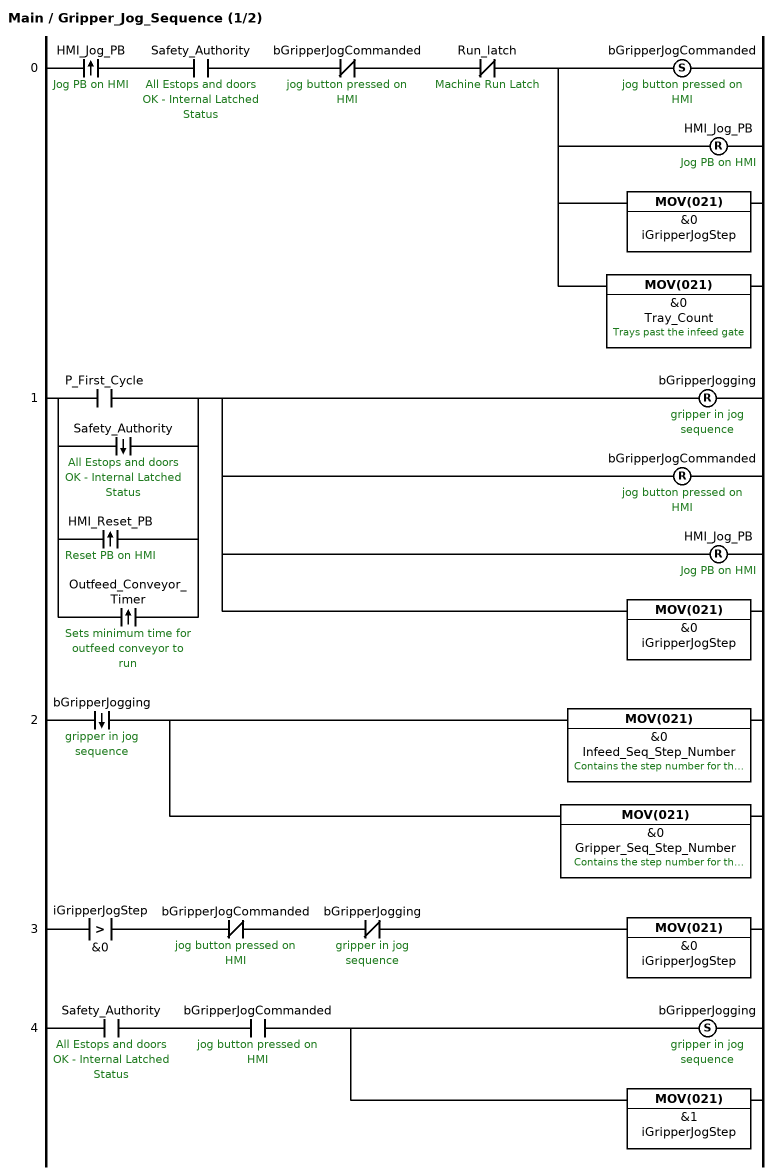
; [picture p144: Main / Gripper_Jog_Sequence, rungs 0-4]
; rung 0
@LD HMI_Jog_PB  ; Jog PB on HMI
AND Safety_Authority  ; All Estops and doors OK - Internal Latched Status
ANDNOT bGripperJogCommanded  ; jog button pressed on HMI
ANDNOT Run_latch  ; Machine Run Latch
SET bGripperJogCommanded  ; jog button pressed on HMI
RSET HMI_Jog_PB  ; Jog PB on HMI
MOV(021) &0 iGripperJogStep
MOV(021) &0 Tray_Count  ; Trays past the infeed gate
; rung 1
LD P_First_Cycle
%OR Safety_Authority  ; All Estops and doors OK - Internal Latched Status
@OR HMI_Reset_PB  ; Reset PB on HMI
@OR Outfeed_Conveyor_Timer  ; Sets minimum time for outfeed conveyor to run
RSET bGripperJogging  ; gripper in jog sequence
RSET bGripperJogCommanded  ; jog button pressed on HMI
RSET HMI_Jog_PB  ; Jog PB on HMI
MOV(021) &0 iGripperJogStep
; rung 2
%LD bGripperJogging  ; gripper in jog sequence
MOV(021) &0 Infeed_Seq_Step_Number  ; Contains the step number for the Infeed sequence
MOV(021) &0 Gripper_Seq_Step_Number  ; Contains the step number for the gripper sequence
; rung 3
LD>(320) iGripperJogStep &0
ANDNOT bGripperJogCommanded  ; jog button pressed on HMI
ANDNOT bGripperJogging  ; gripper in jog sequence
MOV(021) &0 iGripperJogStep
; rung 4
LD Safety_Authority  ; All Estops and doors OK - Internal Latched Status
AND bGripperJogCommanded  ; jog button pressed on HMI
SET bGripperJogging  ; gripper in jog sequence
MOV(021) &1 iGripperJogStep

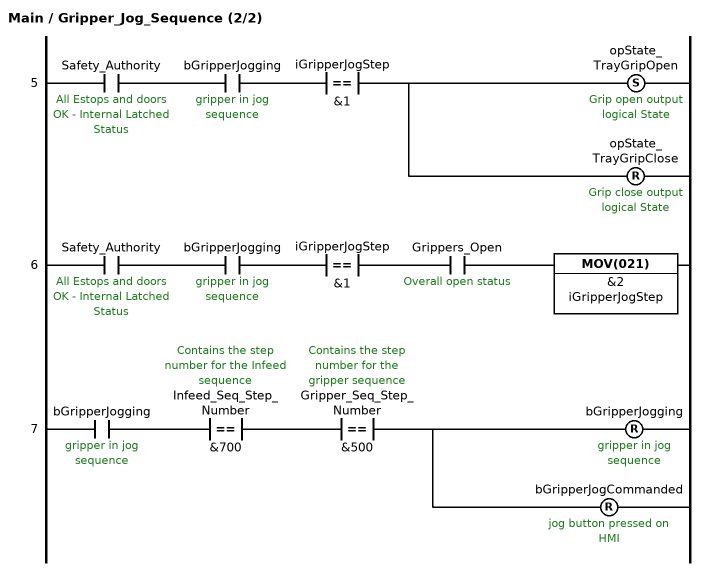
; rung 5
LD Safety_Authority  ; All Estops and doors OK - Internal Latched Status
AND bGripperJogging  ; gripper in jog sequence
AND=(300) iGripperJogStep &1
SET opState_TrayGripOpen  ; Grip open output logical State
RSET opState_TrayGripClose  ; Grip close output logical State
; rung 6
LD Safety_Authority  ; All Estops and doors OK - Internal Latched Status
AND bGripperJogging  ; gripper in jog sequence
AND=(300) iGripperJogStep &1
AND Grippers_Open  ; Overall open status
MOV(021) &2 iGripperJogStep
; rung 7
LD bGripperJogging  ; gripper in jog sequence
AND=(300) Infeed_Seq_Step_Number &700  ; Contains the step number for the Infeed sequence
AND=(300) Gripper_Seq_Step_Number &500  ; Contains the step number for the gripper sequence
RSET bGripperJogging  ; gripper in jog sequence
RSET bGripperJogCommanded  ; jog button pressed on HMI

### Section Machine_Timing

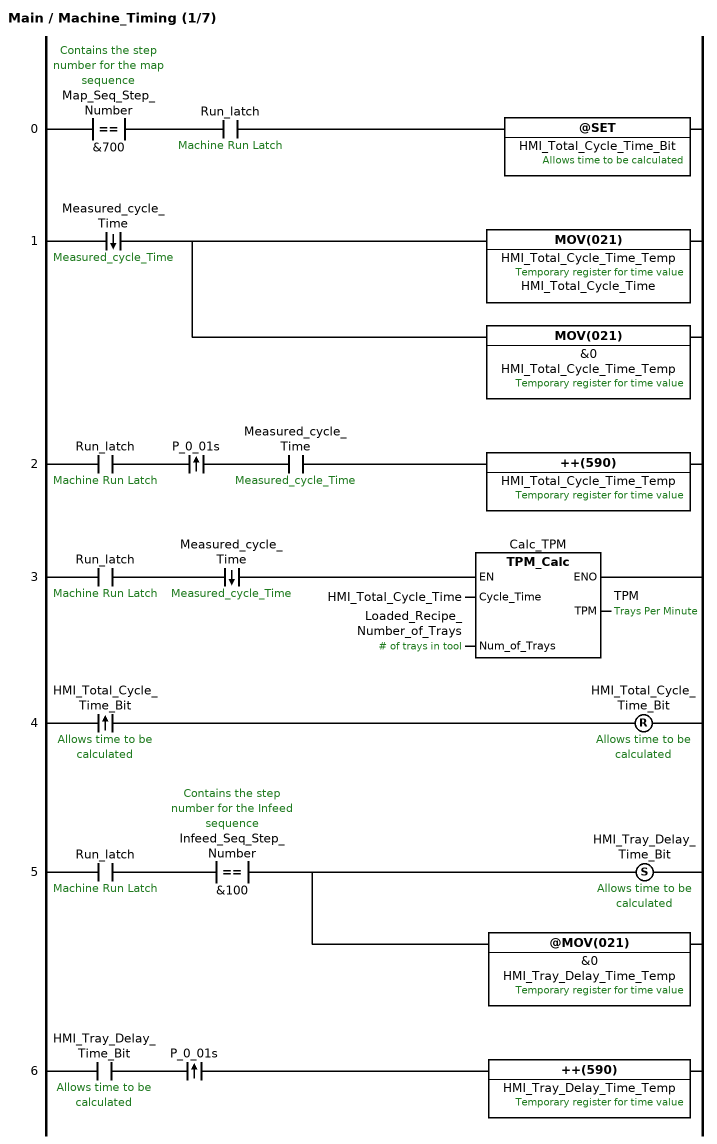
; rung 0
LD=(300) Map_Seq_Step_Number &700  ; Contains the step number for the map sequence
AND Run_latch  ; Machine Run Latch
@SET HMI_Total_Cycle_Time_Bit  ; Allows time to be calculated
; rung 1
%LD Measured_cycle_Time  ; Measured_cycle_Time
MOV(021) HMI_Total_Cycle_Time_Temp HMI_Total_Cycle_Time  ; Temporary register for time value
MOV(021) &0 HMI_Total_Cycle_Time_Temp  ; Temporary register for time value
; rung 2
LD Run_latch  ; Machine Run Latch
@AND P_0_01s
AND Measured_cycle_Time  ; Measured_cycle_Time
++(590) HMI_Total_Cycle_Time_Temp  ; Temporary register for time value
; rung 3
LD Run_latch  ; Machine Run Latch
%AND Measured_cycle_Time  ; Measured_cycle_Time
CALL Calc_TPM : TPM_Calc (Cycle_Time := HMI_Total_Cycle_Time, Num_of_Trays := Loaded_Recipe_Number_of_Trays, TPM => TPM)  ; # of trays in tool, Trays Per Minute
; rung 4
@LD HMI_Total_Cycle_Time_Bit  ; Allows time to be calculated
RSET HMI_Total_Cycle_Time_Bit  ; Allows time to be calculated
; rung 5
LD Run_latch  ; Machine Run Latch
AND=(300) Infeed_Seq_Step_Number &100  ; Contains the step number for the Infeed sequence
SET HMI_Tray_Delay_Time_Bit  ; Allows time to be calculated
@MOV(021) &0 HMI_Tray_Delay_Time_Temp  ; Temporary register for time value
; rung 6
LD HMI_Tray_Delay_Time_Bit  ; Allows time to be calculated
@AND P_0_01s
++(590) HMI_Tray_Delay_Time_Temp  ; Temporary register for time value

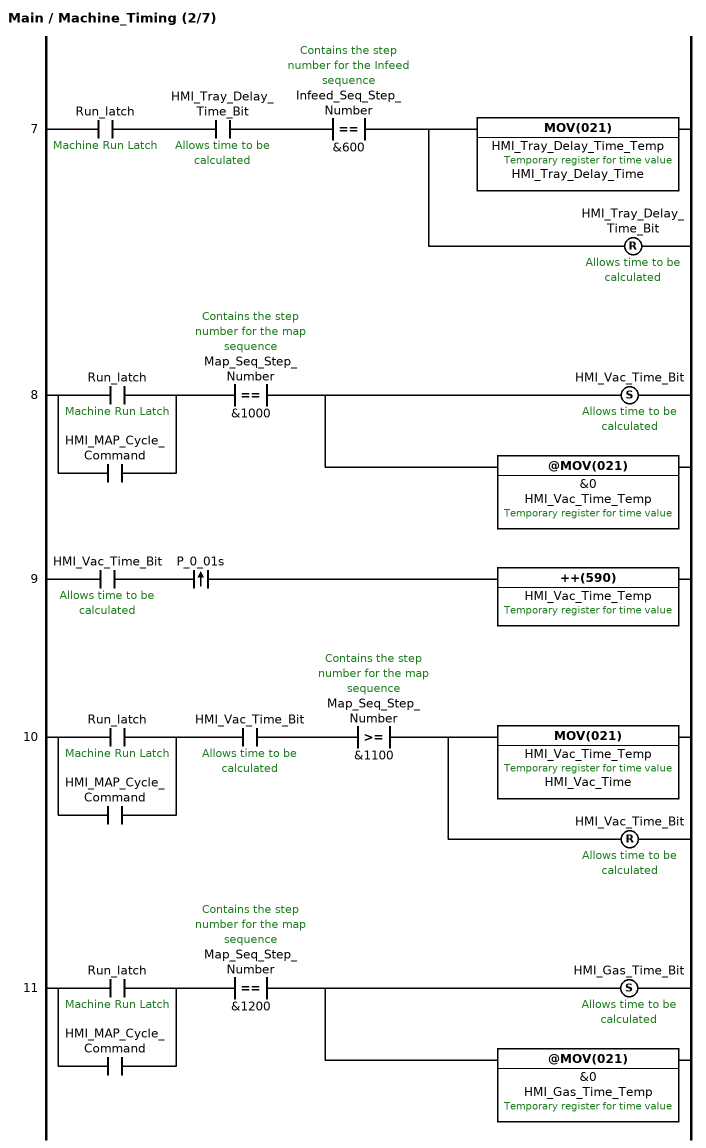
; rung 7
LD Run_latch  ; Machine Run Latch
AND HMI_Tray_Delay_Time_Bit  ; Allows time to be calculated
AND=(300) Infeed_Seq_Step_Number &600  ; Contains the step number for the Infeed sequence
MOV(021) HMI_Tray_Delay_Time_Temp HMI_Tray_Delay_Time  ; Temporary register for time value
RSET HMI_Tray_Delay_Time_Bit  ; Allows time to be calculated
; rung 8
LD Run_latch  ; Machine Run Latch
OR HMI_MAP_Cycle_Command
AND=(300) Map_Seq_Step_Number &1000  ; Contains the step number for the map sequence
SET HMI_Vac_Time_Bit  ; Allows time to be calculated
@MOV(021) &0 HMI_Vac_Time_Temp  ; Temporary register for time value
; rung 9
LD HMI_Vac_Time_Bit  ; Allows time to be calculated
@AND P_0_01s
++(590) HMI_Vac_Time_Temp  ; Temporary register for time value
; rung 10
LD Run_latch  ; Machine Run Latch
OR HMI_MAP_Cycle_Command
AND HMI_Vac_Time_Bit  ; Allows time to be calculated
AND>=(325) Map_Seq_Step_Number &1100  ; Contains the step number for the map sequence
MOV(021) HMI_Vac_Time_Temp HMI_Vac_Time  ; Temporary register for time value
RSET HMI_Vac_Time_Bit  ; Allows time to be calculated
; rung 11
LD Run_latch  ; Machine Run Latch
OR HMI_MAP_Cycle_Command
AND=(300) Map_Seq_Step_Number &1200  ; Contains the step number for the map sequence
SET HMI_Gas_Time_Bit  ; Allows time to be calculated
@MOV(021) &0 HMI_Gas_Time_Temp  ; Temporary register for time value

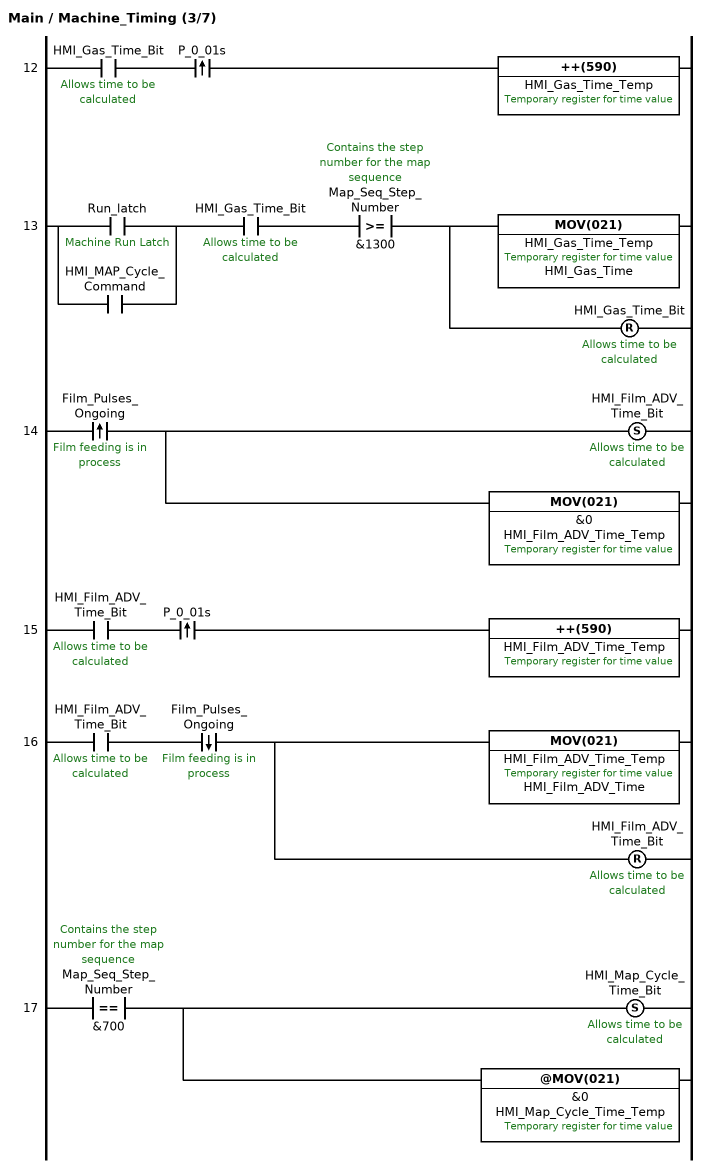
; rung 12
LD HMI_Gas_Time_Bit  ; Allows time to be calculated
@AND P_0_01s
++(590) HMI_Gas_Time_Temp  ; Temporary register for time value
; rung 13
LD Run_latch  ; Machine Run Latch
OR HMI_MAP_Cycle_Command
AND HMI_Gas_Time_Bit  ; Allows time to be calculated
AND>=(325) Map_Seq_Step_Number &1300  ; Contains the step number for the map sequence
MOV(021) HMI_Gas_Time_Temp HMI_Gas_Time  ; Temporary register for time value
RSET HMI_Gas_Time_Bit  ; Allows time to be calculated
; rung 14
@LD Film_Pulses_Ongoing  ; Film feeding is in process
SET HMI_Film_ADV_Time_Bit  ; Allows time to be calculated
MOV(021) &0 HMI_Film_ADV_Time_Temp  ; Temporary register for time value
; rung 15
LD HMI_Film_ADV_Time_Bit  ; Allows time to be calculated
@AND P_0_01s
++(590) HMI_Film_ADV_Time_Temp  ; Temporary register for time value
; rung 16
LD HMI_Film_ADV_Time_Bit  ; Allows time to be calculated
%AND Film_Pulses_Ongoing  ; Film feeding is in process
MOV(021) HMI_Film_ADV_Time_Temp HMI_Film_ADV_Time  ; Temporary register for time value
RSET HMI_Film_ADV_Time_Bit  ; Allows time to be calculated
; rung 17
LD=(300) Map_Seq_Step_Number &700  ; Contains the step number for the map sequence
SET HMI_Map_Cycle_Time_Bit  ; Allows time to be calculated
@MOV(021) &0 HMI_Map_Cycle_Time_Temp  ; Temporary register for time value

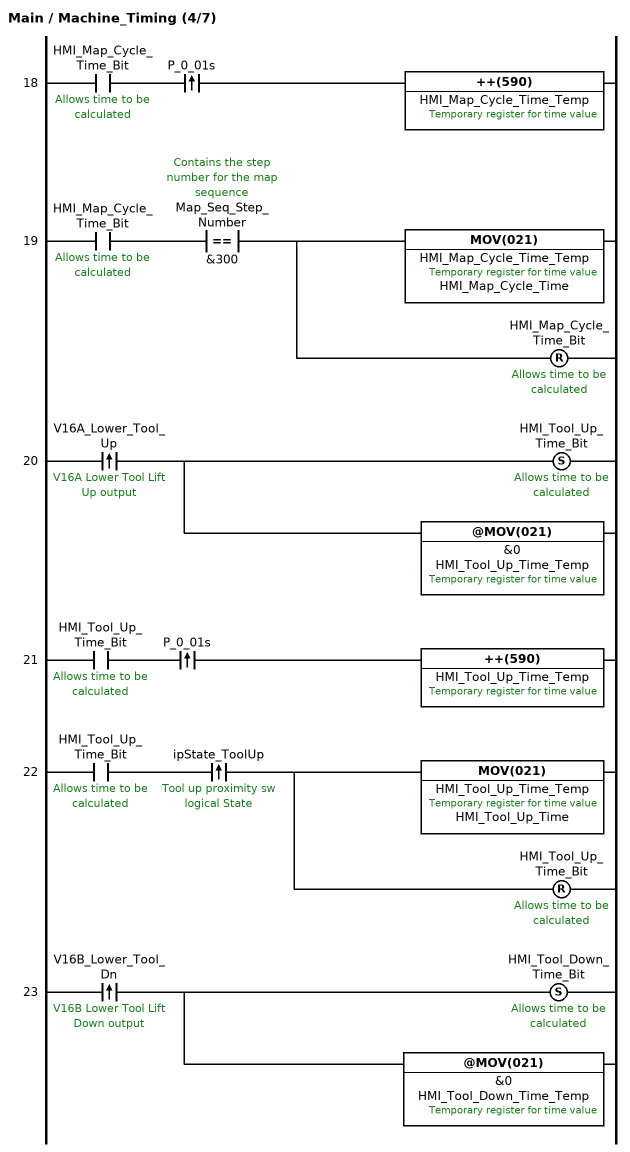
; rung 18
LD HMI_Map_Cycle_Time_Bit  ; Allows time to be calculated
@AND P_0_01s
++(590) HMI_Map_Cycle_Time_Temp  ; Temporary register for time value
; rung 19
LD HMI_Map_Cycle_Time_Bit  ; Allows time to be calculated
AND=(300) Map_Seq_Step_Number &300  ; Contains the step number for the map sequence
MOV(021) HMI_Map_Cycle_Time_Temp HMI_Map_Cycle_Time  ; Temporary register for time value
RSET HMI_Map_Cycle_Time_Bit  ; Allows time to be calculated
; rung 20
@LD V16A_Lower_Tool_Up  ; V16A Lower Tool Lift Up output
SET HMI_Tool_Up_Time_Bit  ; Allows time to be calculated
@MOV(021) &0 HMI_Tool_Up_Time_Temp  ; Temporary register for time value
; rung 21
LD HMI_Tool_Up_Time_Bit  ; Allows time to be calculated
@AND P_0_01s
++(590) HMI_Tool_Up_Time_Temp  ; Temporary register for time value
; rung 22
LD HMI_Tool_Up_Time_Bit  ; Allows time to be calculated
@AND ipState_ToolUp  ; Tool up proximity sw logical State
MOV(021) HMI_Tool_Up_Time_Temp HMI_Tool_Up_Time  ; Temporary register for time value
RSET HMI_Tool_Up_Time_Bit  ; Allows time to be calculated
; rung 23
@LD V16B_Lower_Tool_Dn  ; V16B Lower Tool Lift Down output
SET HMI_Tool_Down_Time_Bit  ; Allows time to be calculated
@MOV(021) &0 HMI_Tool_Down_Time_Temp  ; Temporary register for time value

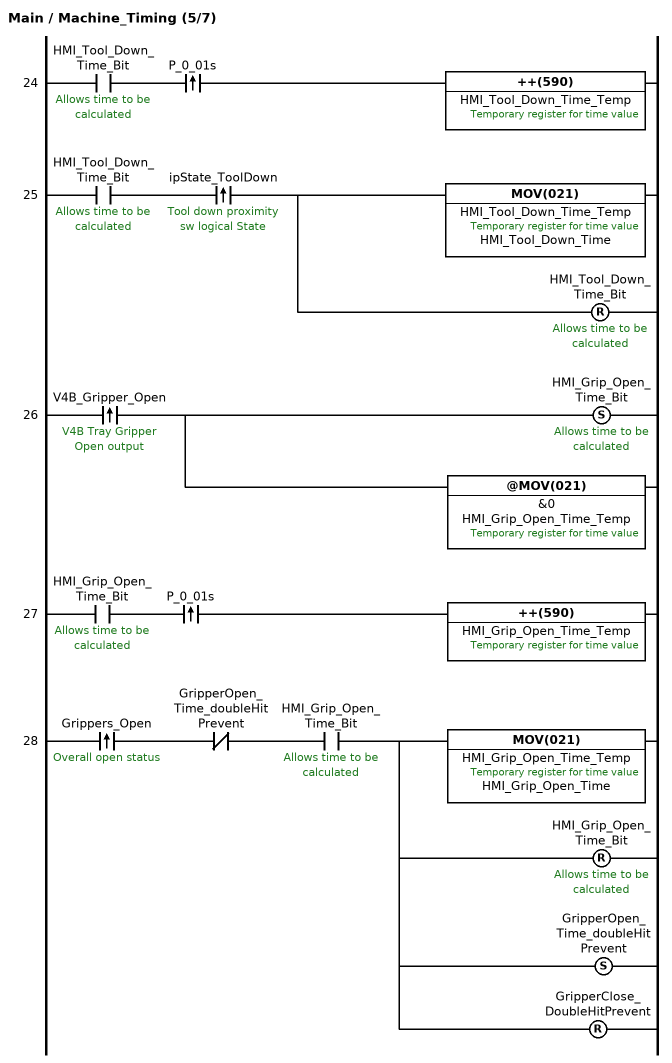
; rung 24
LD HMI_Tool_Down_Time_Bit  ; Allows time to be calculated
@AND P_0_01s
++(590) HMI_Tool_Down_Time_Temp  ; Temporary register for time value
; rung 25
LD HMI_Tool_Down_Time_Bit  ; Allows time to be calculated
@AND ipState_ToolDown  ; Tool down proximity sw logical State
MOV(021) HMI_Tool_Down_Time_Temp HMI_Tool_Down_Time  ; Temporary register for time value
RSET HMI_Tool_Down_Time_Bit  ; Allows time to be calculated
; rung 26
@LD V4B_Gripper_Open  ; V4B Tray Gripper Open output
SET HMI_Grip_Open_Time_Bit  ; Allows time to be calculated
@MOV(021) &0 HMI_Grip_Open_Time_Temp  ; Temporary register for time value
; rung 27
LD HMI_Grip_Open_Time_Bit  ; Allows time to be calculated
@AND P_0_01s
++(590) HMI_Grip_Open_Time_Temp  ; Temporary register for time value
; rung 28
@LD Grippers_Open  ; Overall open status
ANDNOT GripperOpen_Time_doubleHitPrevent
AND HMI_Grip_Open_Time_Bit  ; Allows time to be calculated
MOV(021) HMI_Grip_Open_Time_Temp HMI_Grip_Open_Time  ; Temporary register for time value
RSET HMI_Grip_Open_Time_Bit  ; Allows time to be calculated
SET GripperOpen_Time_doubleHitPrevent
RSET GripperClose_DoubleHitPrevent

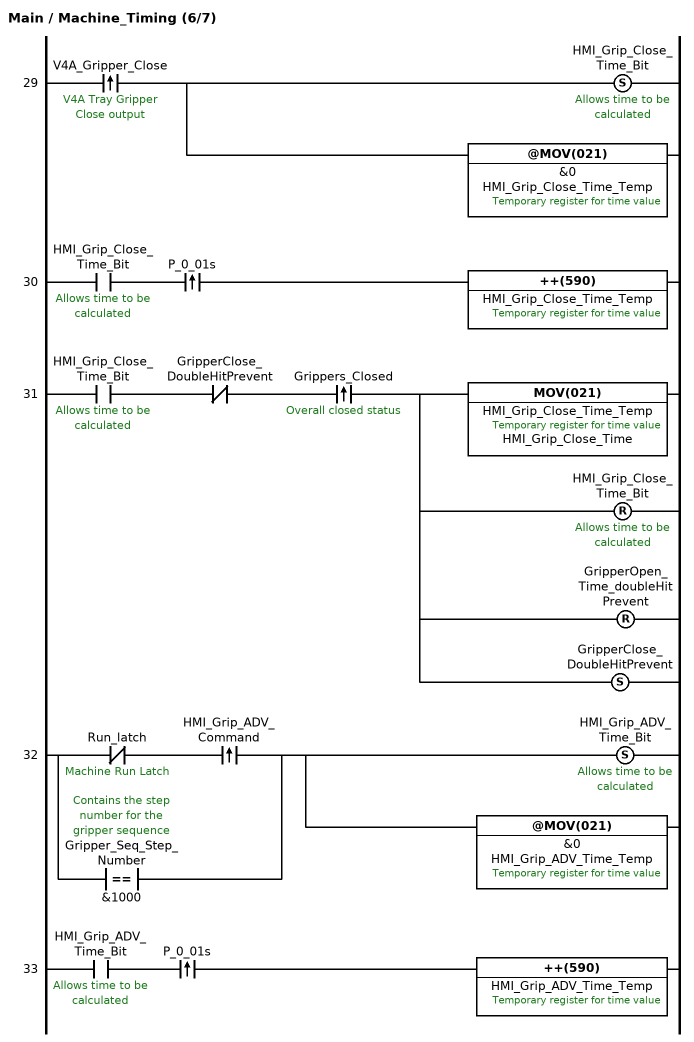
; rung 29
@LD V4A_Gripper_Close  ; V4A Tray Gripper Close output
SET HMI_Grip_Close_Time_Bit  ; Allows time to be calculated
@MOV(021) &0 HMI_Grip_Close_Time_Temp  ; Temporary register for time value
; rung 30
LD HMI_Grip_Close_Time_Bit  ; Allows time to be calculated
@AND P_0_01s
++(590) HMI_Grip_Close_Time_Temp  ; Temporary register for time value
; rung 31
LD HMI_Grip_Close_Time_Bit  ; Allows time to be calculated
ANDNOT GripperClose_DoubleHitPrevent
@AND Grippers_Closed  ; Overall closed status
MOV(021) HMI_Grip_Close_Time_Temp HMI_Grip_Close_Time  ; Temporary register for time value
RSET HMI_Grip_Close_Time_Bit  ; Allows time to be calculated
RSET GripperOpen_Time_doubleHitPrevent
SET GripperClose_DoubleHitPrevent
; rung 32
LDNOT Run_latch  ; Machine Run Latch
@AND HMI_Grip_ADV_Command
OR=(300) Gripper_Seq_Step_Number &1000  ; Contains the step number for the gripper sequence
SET HMI_Grip_ADV_Time_Bit  ; Allows time to be calculated
@MOV(021) &0 HMI_Grip_ADV_Time_Temp  ; Temporary register for time value
; rung 33
LD HMI_Grip_ADV_Time_Bit  ; Allows time to be calculated
@AND P_0_01s
++(590) HMI_Grip_ADV_Time_Temp  ; Temporary register for time value

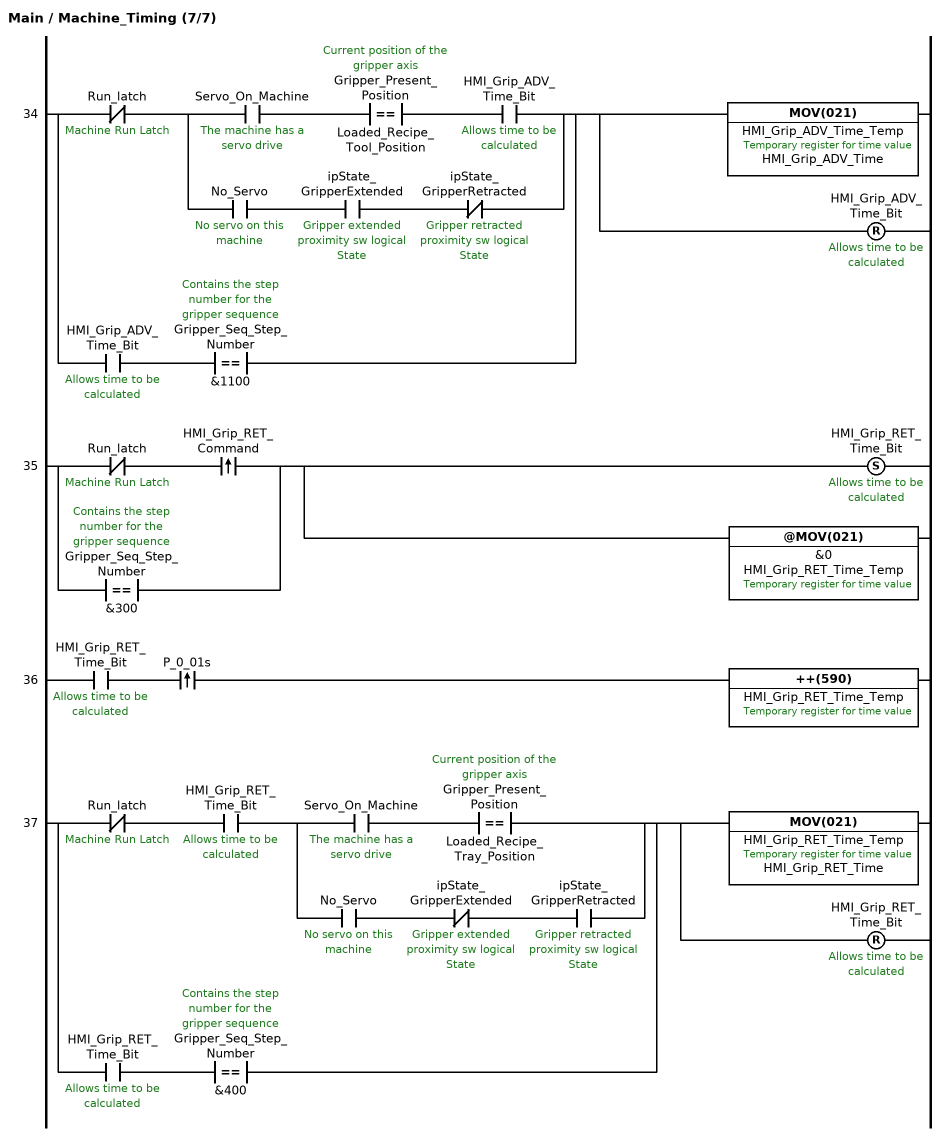
; rung 34
LDNOT Run_latch  ; Machine Run Latch
LD Servo_On_Machine  ; The machine has a servo drive
AND=(300) Gripper_Present_Position Loaded_Recipe_Tool_Position  ; Current position of the gripper axis
AND HMI_Grip_ADV_Time_Bit  ; Allows time to be calculated
LD No_Servo  ; No servo on this machine
AND ipState_GripperExtended  ; Gripper extended proximity sw logical State
ANDNOT ipState_GripperRetracted  ; Gripper retracted proximity sw logical State
ORLD
ANDLD
LD HMI_Grip_ADV_Time_Bit  ; Allows time to be calculated
AND=(300) Gripper_Seq_Step_Number &1100  ; Contains the step number for the gripper sequence
ORLD
MOV(021) HMI_Grip_ADV_Time_Temp HMI_Grip_ADV_Time  ; Temporary register for time value
RSET HMI_Grip_ADV_Time_Bit  ; Allows time to be calculated
; rung 35
LDNOT Run_latch  ; Machine Run Latch
@AND HMI_Grip_RET_Command
OR=(300) Gripper_Seq_Step_Number &300  ; Contains the step number for the gripper sequence
SET HMI_Grip_RET_Time_Bit  ; Allows time to be calculated
@MOV(021) &0 HMI_Grip_RET_Time_Temp  ; Temporary register for time value
; rung 36
LD HMI_Grip_RET_Time_Bit  ; Allows time to be calculated
@AND P_0_01s
++(590) HMI_Grip_RET_Time_Temp  ; Temporary register for time value
; rung 37
LDNOT Run_latch  ; Machine Run Latch
AND HMI_Grip_RET_Time_Bit  ; Allows time to be calculated
LD Servo_On_Machine  ; The machine has a servo drive
AND=(300) Gripper_Present_Position Loaded_Recipe_Tray_Position  ; Current position of the gripper axis
LD No_Servo  ; No servo on this machine
ANDNOT ipState_GripperExtended  ; Gripper extended proximity sw logical State
AND ipState_GripperRetracted  ; Gripper retracted proximity sw logical State
ORLD
ANDLD
LD HMI_Grip_RET_Time_Bit  ; Allows time to be calculated
AND=(300) Gripper_Seq_Step_Number &400  ; Contains the step number for the gripper sequence
ORLD
MOV(021) HMI_Grip_RET_Time_Temp HMI_Grip_RET_Time  ; Temporary register for time value
RSET HMI_Grip_RET_Time_Bit  ; Allows time to be calculated

### Section Vacuum_Test

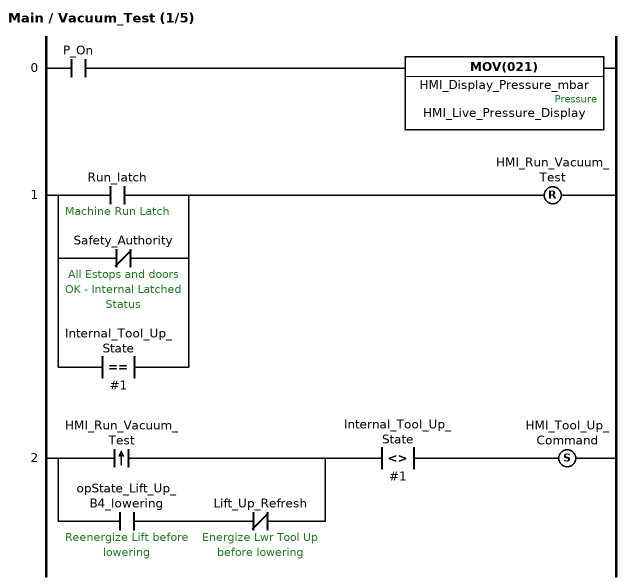
; rung 0
LD P_On
MOV(021) HMI_Display_Pressure_mbar HMI_Live_Pressure_Display  ; Pressure
; rung 1
LD Run_latch  ; Machine Run Latch
ORNOT Safety_Authority  ; All Estops and doors OK - Internal Latched Status
OR=(300) Internal_Tool_Up_State #1
RSET HMI_Run_Vacuum_Test
; rung 2
@LD HMI_Run_Vacuum_Test
LD opState_Lift_Up_B4_lowering  ; Reenergize Lift before lowering
ANDNOT Lift_Up_Refresh  ; Energize Lwr Tool Up before lowering
ORLD
AND<>(305) Internal_Tool_Up_State #1
SET HMI_Tool_Up_Command

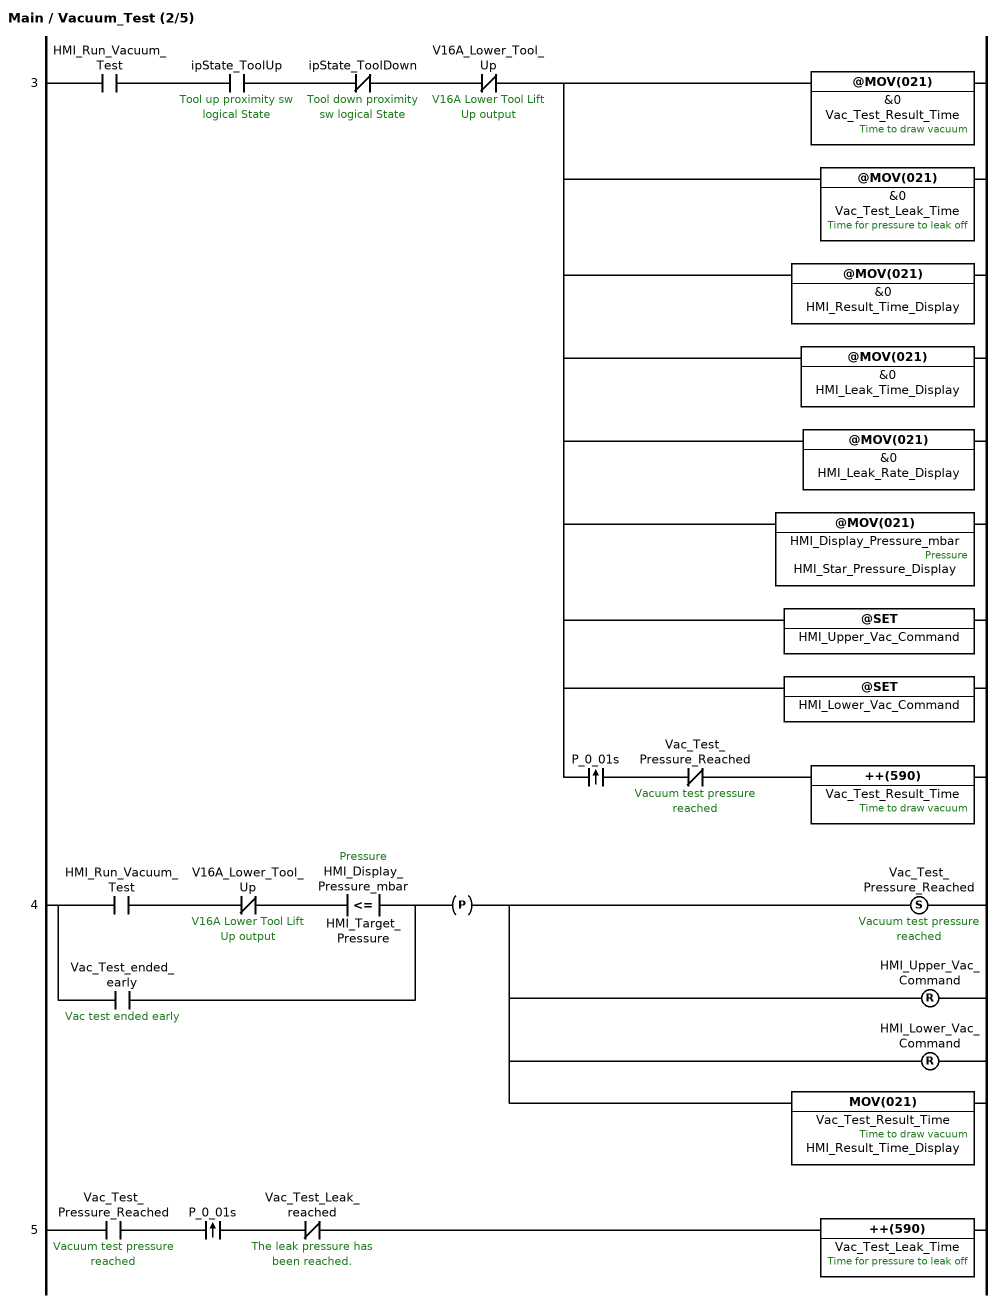
; rung 3
LD HMI_Run_Vacuum_Test
AND ipState_ToolUp  ; Tool up proximity sw logical State
ANDNOT ipState_ToolDown  ; Tool down proximity sw logical State
ANDNOT V16A_Lower_Tool_Up  ; V16A Lower Tool Lift Up output
@MOV(021) &0 Vac_Test_Result_Time  ; Time to draw vacuum
@MOV(021) &0 Vac_Test_Leak_Time  ; Time for pressure to leak off
@MOV(021) &0 HMI_Result_Time_Display
@MOV(021) &0 HMI_Leak_Time_Display
@MOV(021) &0 HMI_Leak_Rate_Display
@MOV(021) HMI_Display_Pressure_mbar HMI_Star_Pressure_Display  ; Pressure
@SET HMI_Upper_Vac_Command
@SET HMI_Lower_Vac_Command
@AND P_0_01s
ANDNOT Vac_Test_Pressure_Reached  ; Vacuum test pressure reached
++(590) Vac_Test_Result_Time  ; Time to draw vacuum
; rung 4
LD HMI_Run_Vacuum_Test
ANDNOT V16A_Lower_Tool_Up  ; V16A Lower Tool Lift Up output
AND<=(315) HMI_Display_Pressure_mbar HMI_Target_Pressure  ; Pressure
OR Vac_Test_ended_early  ; Vac test ended early
UP(521)
SET Vac_Test_Pressure_Reached  ; Vacuum test pressure reached
RSET HMI_Upper_Vac_Command
RSET HMI_Lower_Vac_Command
MOV(021) Vac_Test_Result_Time HMI_Result_Time_Display  ; Time to draw vacuum
; rung 5
LD Vac_Test_Pressure_Reached  ; Vacuum test pressure reached
@AND P_0_01s
ANDNOT Vac_Test_Leak_reached  ; The leak pressure has been reached.
++(590) Vac_Test_Leak_Time  ; Time for pressure to leak off

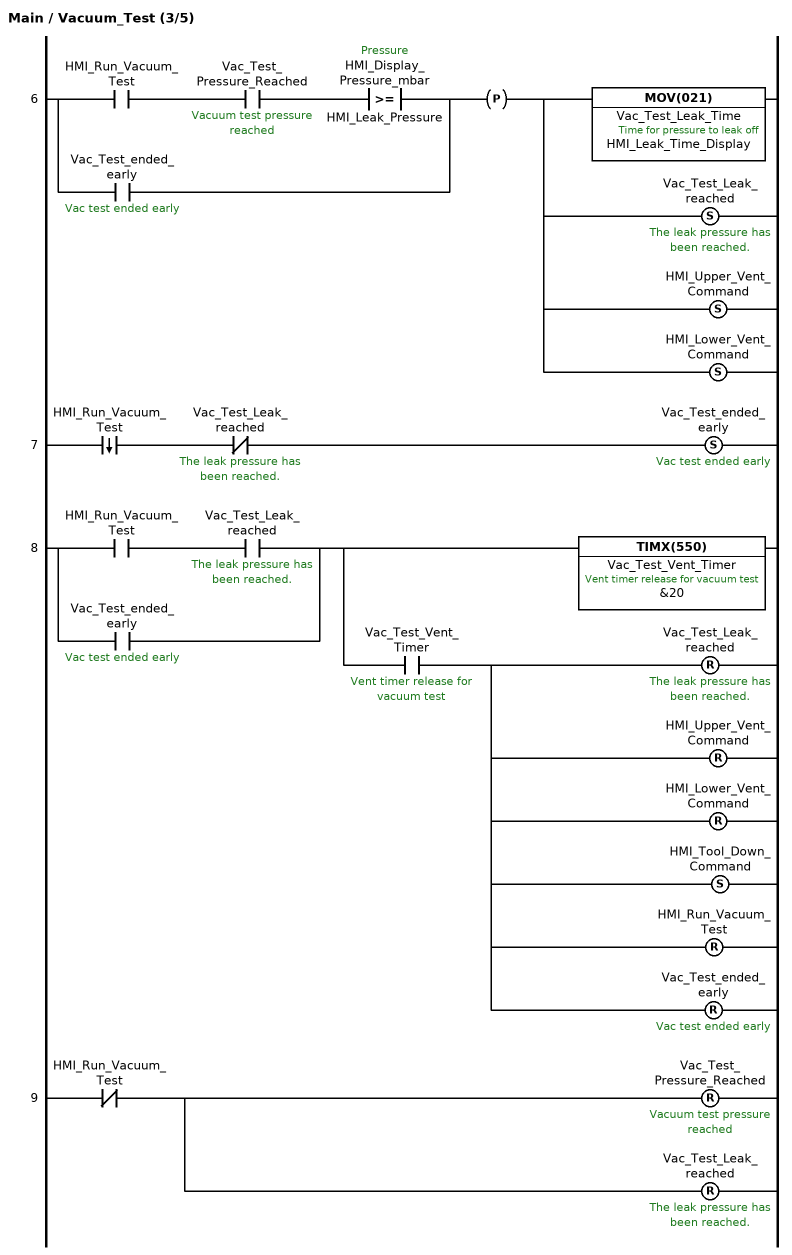
; rung 6
LD HMI_Run_Vacuum_Test
AND Vac_Test_Pressure_Reached  ; Vacuum test pressure reached
AND>=(325) HMI_Display_Pressure_mbar HMI_Leak_Pressure  ; Pressure
OR Vac_Test_ended_early  ; Vac test ended early
UP(521)
MOV(021) Vac_Test_Leak_Time HMI_Leak_Time_Display  ; Time for pressure to leak off
SET Vac_Test_Leak_reached  ; The leak pressure has been reached.
SET HMI_Upper_Vent_Command
SET HMI_Lower_Vent_Command
; rung 7
%LD HMI_Run_Vacuum_Test
ANDNOT Vac_Test_Leak_reached  ; The leak pressure has been reached.
SET Vac_Test_ended_early  ; Vac test ended early
; rung 8
LD HMI_Run_Vacuum_Test
AND Vac_Test_Leak_reached  ; The leak pressure has been reached.
OR Vac_Test_ended_early  ; Vac test ended early
TIMX(550) Vac_Test_Vent_Timer &20  ; Vent timer release for vacuum test
AND Vac_Test_Vent_Timer  ; Vent timer release for vacuum test
RSET Vac_Test_Leak_reached  ; The leak pressure has been reached.
RSET HMI_Upper_Vent_Command
RSET HMI_Lower_Vent_Command
SET HMI_Tool_Down_Command
RSET HMI_Run_Vacuum_Test
RSET Vac_Test_ended_early  ; Vac test ended early
; rung 9
LDNOT HMI_Run_Vacuum_Test
RSET Vac_Test_Pressure_Reached  ; Vacuum test pressure reached
RSET Vac_Test_Leak_reached  ; The leak pressure has been reached.

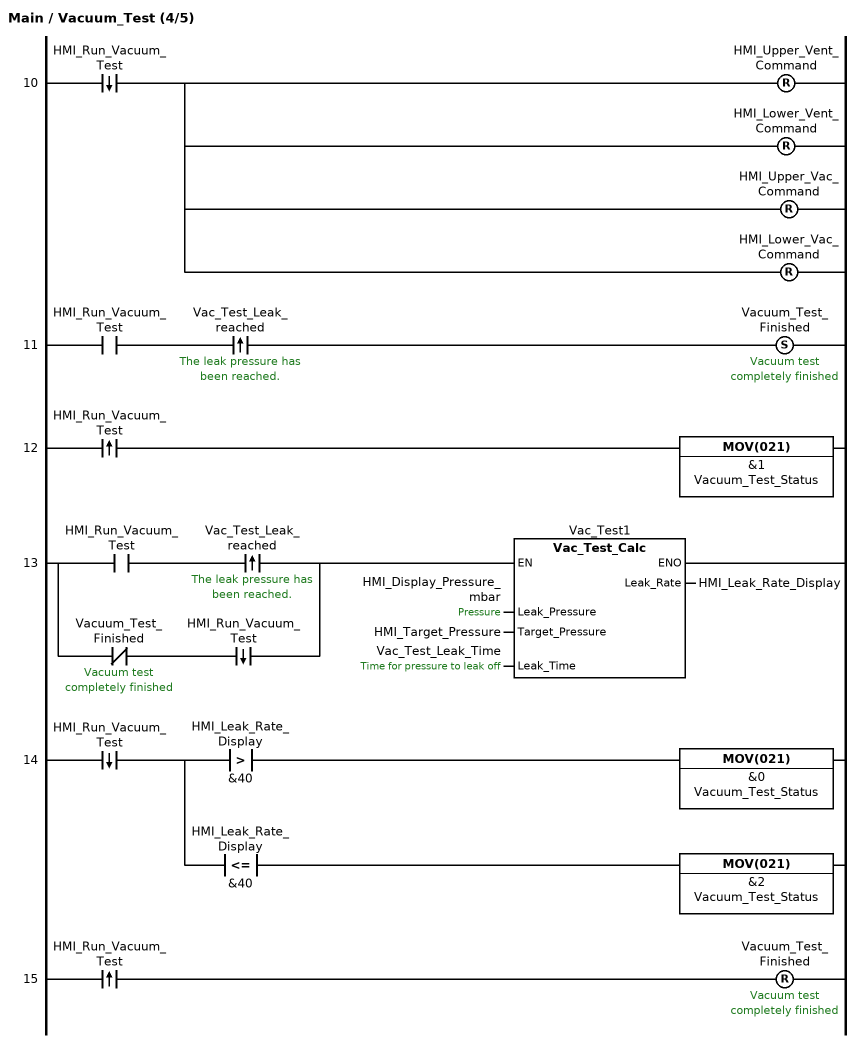
; rung 10
%LD HMI_Run_Vacuum_Test
RSET HMI_Upper_Vent_Command
RSET HMI_Lower_Vent_Command
RSET HMI_Upper_Vac_Command
RSET HMI_Lower_Vac_Command
; rung 11
LD HMI_Run_Vacuum_Test
@AND Vac_Test_Leak_reached  ; The leak pressure has been reached.
SET Vacuum_Test_Finished  ; Vacuum test completely finished
; rung 12
@LD HMI_Run_Vacuum_Test
MOV(021) &1 Vacuum_Test_Status
; rung 13
LD HMI_Run_Vacuum_Test
@AND Vac_Test_Leak_reached  ; The leak pressure has been reached.
LDNOT Vacuum_Test_Finished  ; Vacuum test completely finished
%AND HMI_Run_Vacuum_Test
ORLD
CALL Vac_Test1 : Vac_Test_Calc (Leak_Pressure := HMI_Display_Pressure_mbar, Target_Pressure := HMI_Target_Pressure, Leak_Time := Vac_Test_Leak_Time, Leak_Rate => HMI_Leak_Rate_Display)  ; Pressure, Time for pressure to leak off
; rung 14
%LD HMI_Run_Vacuum_Test
OUT TR0
AND>(320) HMI_Leak_Rate_Display &40
MOV(021) &0 Vacuum_Test_Status
LD TR0
AND<=(315) HMI_Leak_Rate_Display &40
MOV(021) &2 Vacuum_Test_Status
; rung 15
@LD HMI_Run_Vacuum_Test
RSET Vacuum_Test_Finished  ; Vacuum test completely finished

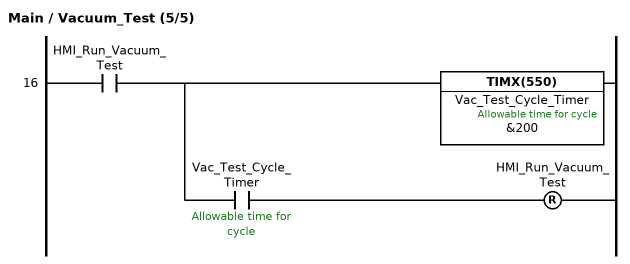
; rung 16
LD HMI_Run_Vacuum_Test
TIMX(550) Vac_Test_Cycle_Timer &200  ; Allowable time for cycle
AND Vac_Test_Cycle_Timer  ; Allowable time for cycle
RSET HMI_Run_Vacuum_Test

### Section HMI

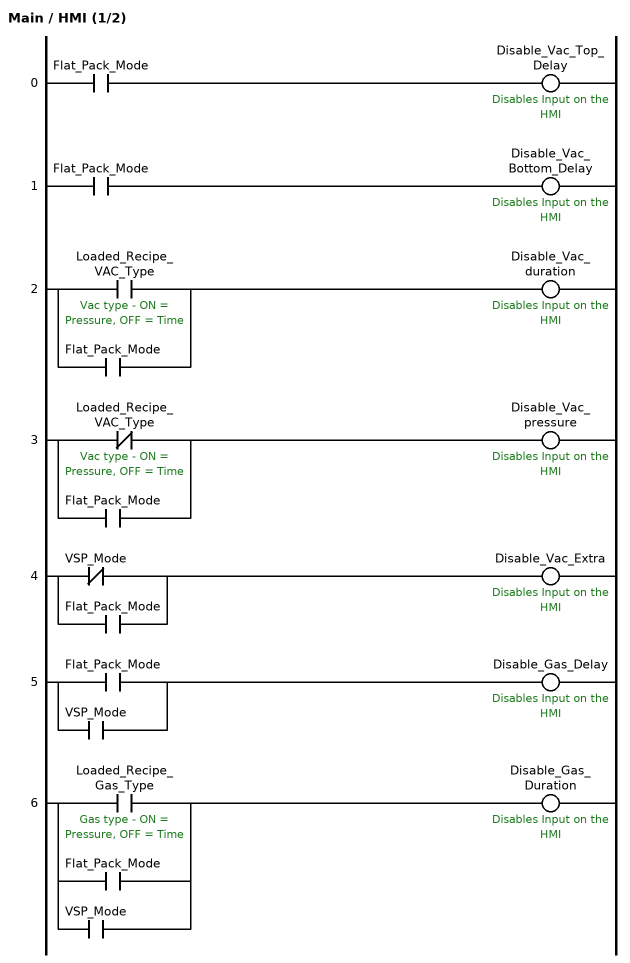
; rung 0
LD Flat_Pack_Mode
OUT Disable_Vac_Top_Delay  ; Disables Input on the HMI
; rung 1
LD Flat_Pack_Mode
OUT Disable_Vac_Bottom_Delay  ; Disables Input on the HMI
; rung 2
LD Loaded_Recipe_VAC_Type  ; Vac type - ON = Pressure, OFF = Time
OR Flat_Pack_Mode
OUT Disable_Vac_duration  ; Disables Input on the HMI
; rung 3
LDNOT Loaded_Recipe_VAC_Type  ; Vac type - ON = Pressure, OFF = Time
OR Flat_Pack_Mode
OUT Disable_Vac_pressure  ; Disables Input on the HMI
; rung 4
LDNOT VSP_Mode
OR Flat_Pack_Mode
OUT Disable_Vac_Extra  ; Disables Input on the HMI
; rung 5
LD Flat_Pack_Mode
OR VSP_Mode
OUT Disable_Gas_Delay  ; Disables Input on the HMI
; rung 6
LD Loaded_Recipe_Gas_Type  ; Gas type - ON = Pressure, OFF = Time
OR Flat_Pack_Mode
OR VSP_Mode
OUT Disable_Gas_Duration  ; Disables Input on the HMI

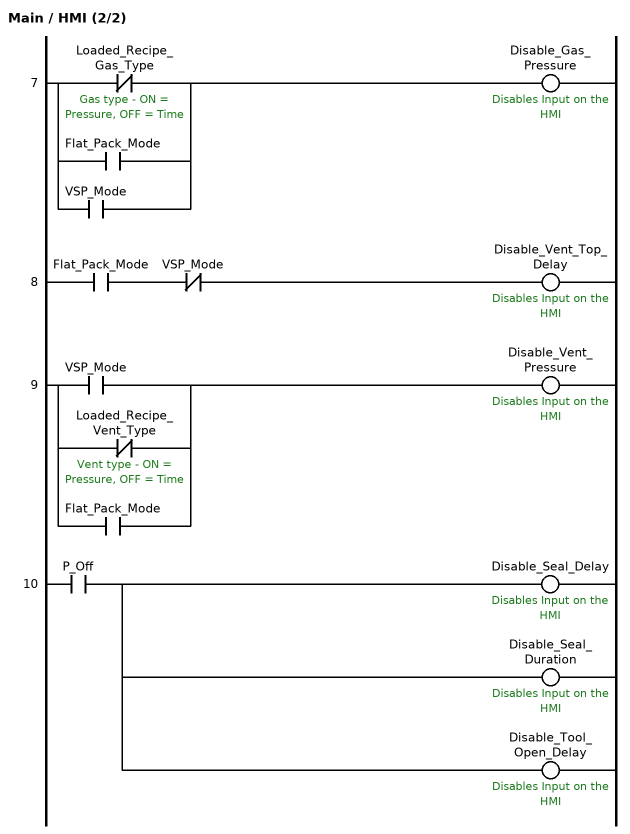
; rung 7
LDNOT Loaded_Recipe_Gas_Type  ; Gas type - ON = Pressure, OFF = Time
OR Flat_Pack_Mode
OR VSP_Mode
OUT Disable_Gas_Pressure  ; Disables Input on the HMI
; rung 8
LD Flat_Pack_Mode
ANDNOT VSP_Mode
OUT Disable_Vent_Top_Delay  ; Disables Input on the HMI
; rung 9
LD VSP_Mode
ORNOT Loaded_Recipe_Vent_Type  ; Vent type - ON = Pressure, OFF = Time
OR Flat_Pack_Mode
OUT Disable_Vent_Pressure  ; Disables Input on the HMI
; rung 10
LD P_Off
OUT Disable_Seal_Delay  ; Disables Input on the HMI
OUT Disable_Seal_Duration  ; Disables Input on the HMI
OUT Disable_Tool_Open_Delay  ; Disables Input on the HMI

### Section Vacuum_Graph

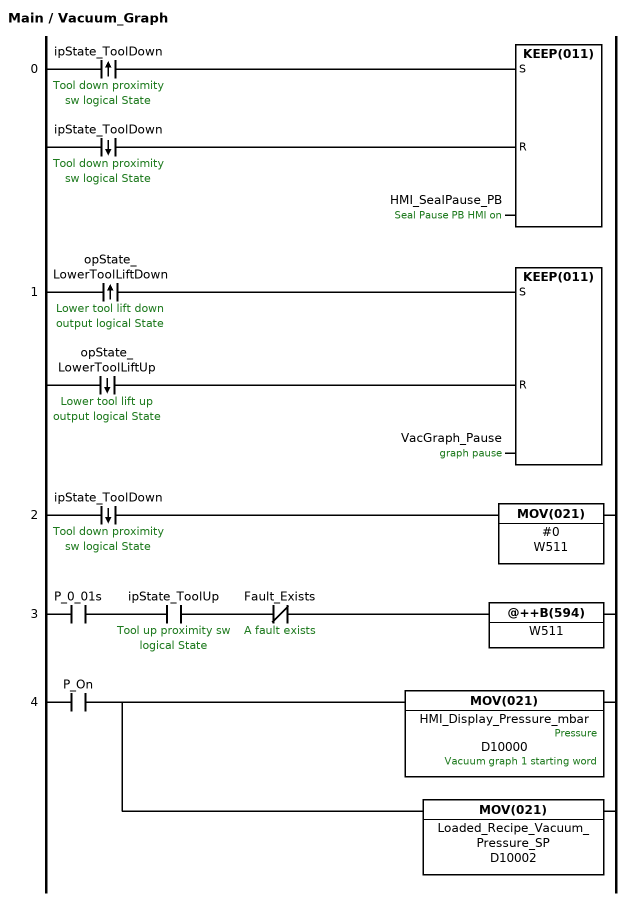
; rung 0
@LD ipState_ToolDown  ; Tool down proximity sw logical State
%LD ipState_ToolDown  ; Tool down proximity sw logical State
KEEP(011) HMI_SealPause_PB  ; Seal Pause PB HMI on
; rung 1
@LD opState_LowerToolLiftDown  ; Lower tool lift down output logical State
%LD opState_LowerToolLiftUp  ; Lower tool lift up output logical State
KEEP(011) VacGraph_Pause  ; graph pause
; rung 2
%LD ipState_ToolDown  ; Tool down proximity sw logical State
MOV(021) #0 W511
; rung 3
LD P_0_01s
AND ipState_ToolUp  ; Tool up proximity sw logical State
ANDNOT Fault_Exists  ; A fault exists
@++B(594) W511
; rung 4
LD P_On
MOV(021) HMI_Display_Pressure_mbar D10000  ; Pressure, Vacuum graph 1 starting word
MOV(021) Loaded_Recipe_Vacuum_Pressure_SP D10002

### Section PopUp

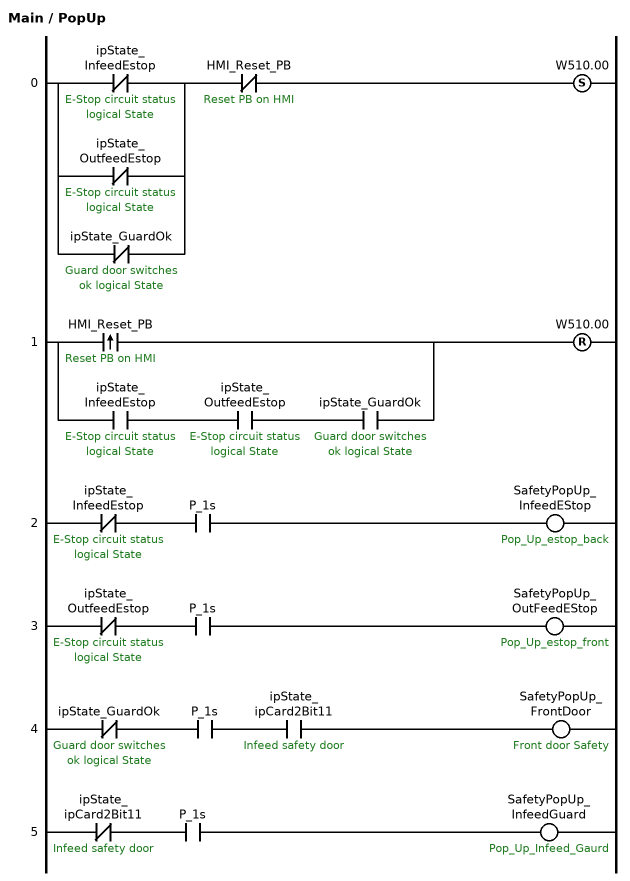
; rung 0
LDNOT ipState_InfeedEstop  ; E-Stop circuit status logical State
ORNOT ipState_OutfeedEstop  ; E-Stop circuit status logical State
ORNOT ipState_GuardOk  ; Guard door switches ok logical State
ANDNOT HMI_Reset_PB  ; Reset PB on HMI
SET W510.00
; rung 1
@LD HMI_Reset_PB  ; Reset PB on HMI
LD ipState_InfeedEstop  ; E-Stop circuit status logical State
AND ipState_OutfeedEstop  ; E-Stop circuit status logical State
AND ipState_GuardOk  ; Guard door switches ok logical State
ORLD
RSET W510.00
; rung 2
LDNOT ipState_InfeedEstop  ; E-Stop circuit status logical State
AND P_1s
OUT SafetyPopUp_InfeedEStop  ; Pop_Up_estop_back
; rung 3
LDNOT ipState_OutfeedEstop  ; E-Stop circuit status logical State
AND P_1s
OUT SafetyPopUp_OutFeedEStop  ; Pop_Up_estop_front
; rung 4
LDNOT ipState_GuardOk  ; Guard door switches ok logical State
AND P_1s
AND ipState_ipCard2Bit11  ; Infeed safety door
OUT SafetyPopUp_FrontDoor  ; Front door Safety
; rung 5
LDNOT ipState_ipCard2Bit11  ; Infeed safety door
AND P_1s
OUT SafetyPopUp_InfeedGuard  ; Pop_Up_Infeed_Gaurd

### Section UPSTREAM_CONV__GATE

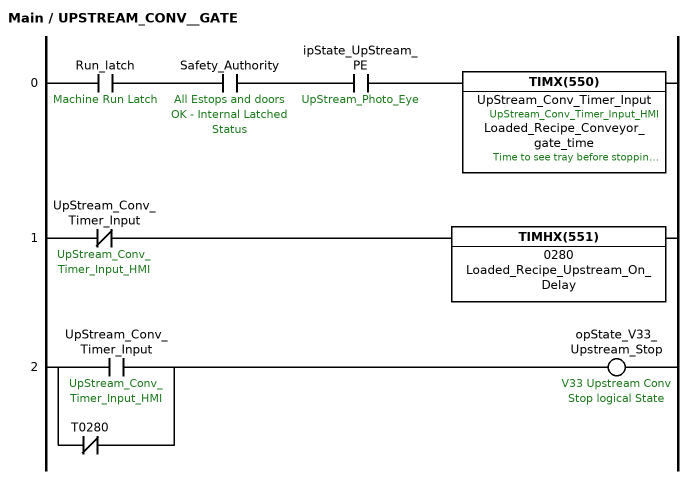
; rung 0
LD Run_latch  ; Machine Run Latch
AND Safety_Authority  ; All Estops and doors OK - Internal Latched Status
AND ipState_UpStream_PE  ; UpStream_Photo_Eye
TIMX(550) UpStream_Conv_Timer_Input Loaded_Recipe_Conveyor_gate_time  ; UpStream_Conv_Timer_Input_HMI, Time to see tray before stopping upstream
; rung 1
LDNOT UpStream_Conv_Timer_Input  ; UpStream_Conv_Timer_Input_HMI
TIMHX(551) 0280 Loaded_Recipe_Upstream_On_Delay
; rung 2
LD UpStream_Conv_Timer_Input  ; UpStream_Conv_Timer_Input_HMI
ORNOT T0280
OUT opState_V33_Upstream_Stop  ; V33 Upstream Conv Stop logical State

### Section END
; rung 0
END(001)

## Program Temp_CNTR (cyclic task 20)

### Section TC102_12
; Unit 02, Input type 0, Dipswitch 1-2-3-4-5-6-7 Off,  8 On

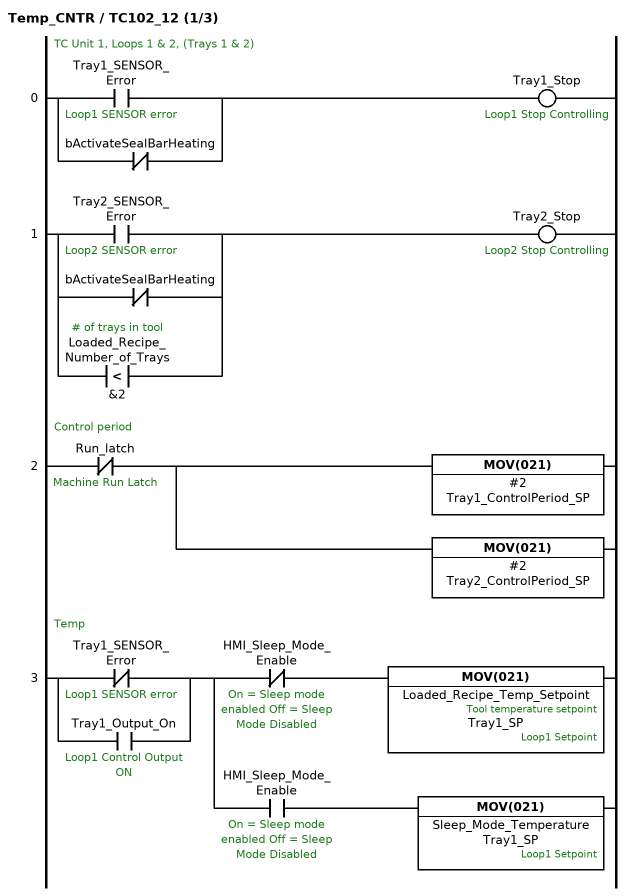
; rung 0: TC Unit 1, Loops 1 & 2, (Trays 1 & 2)
LD Tray1_SENSOR_Error  ; Loop1 SENSOR error
ORNOT bActivateSealBarHeating
OUT Tray1_Stop  ; Loop1 Stop Controlling
; rung 1
LD Tray2_SENSOR_Error  ; Loop2 SENSOR error
ORNOT bActivateSealBarHeating
OR<(310) Loaded_Recipe_Number_of_Trays &2  ; # of trays in tool
OUT Tray2_Stop  ; Loop2 Stop Controlling
; rung 2: Control period
LDNOT Run_latch  ; Machine Run Latch
MOV(021) #2 Tray1_ControlPeriod_SP
MOV(021) #2 Tray2_ControlPeriod_SP
; rung 3: Temp
LDNOT Tray1_SENSOR_Error  ; Loop1 SENSOR error
OR Tray1_Output_On  ; Loop1 Control Output ON
OUT TR0
ANDNOT HMI_Sleep_Mode_Enable  ; On = Sleep mode enabled Off = Sleep Mode Disabled
MOV(021) Loaded_Recipe_Temp_Setpoint Tray1_SP  ; Tool temperature setpoint, Loop1 Setpoint
LD TR0
AND HMI_Sleep_Mode_Enable  ; On = Sleep mode enabled Off = Sleep Mode Disabled
MOV(021) Sleep_Mode_Temperature Tray1_SP  ; Loop1 Setpoint

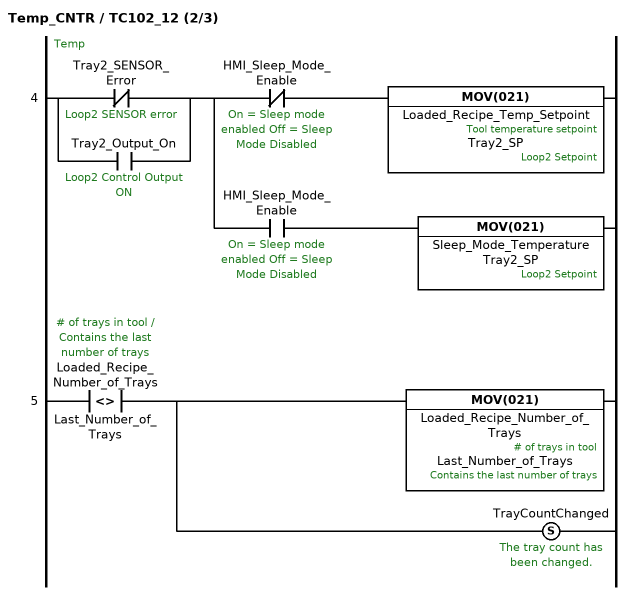
; rung 4: Temp
LDNOT Tray2_SENSOR_Error  ; Loop2 SENSOR error
OR Tray2_Output_On  ; Loop2 Control Output ON
OUT TR0
ANDNOT HMI_Sleep_Mode_Enable  ; On = Sleep mode enabled Off = Sleep Mode Disabled
MOV(021) Loaded_Recipe_Temp_Setpoint Tray2_SP  ; Tool temperature setpoint, Loop2 Setpoint
LD TR0
AND HMI_Sleep_Mode_Enable  ; On = Sleep mode enabled Off = Sleep Mode Disabled
MOV(021) Sleep_Mode_Temperature Tray2_SP  ; Loop2 Setpoint
; rung 5
LD<>(305) Loaded_Recipe_Number_of_Trays Last_Number_of_Trays  ; # of trays in tool, Contains the last number of trays
MOV(021) Loaded_Recipe_Number_of_Trays Last_Number_of_Trays  ; # of trays in tool, Contains the last number of trays
SET TrayCountChanged  ; The tray count has been changed.

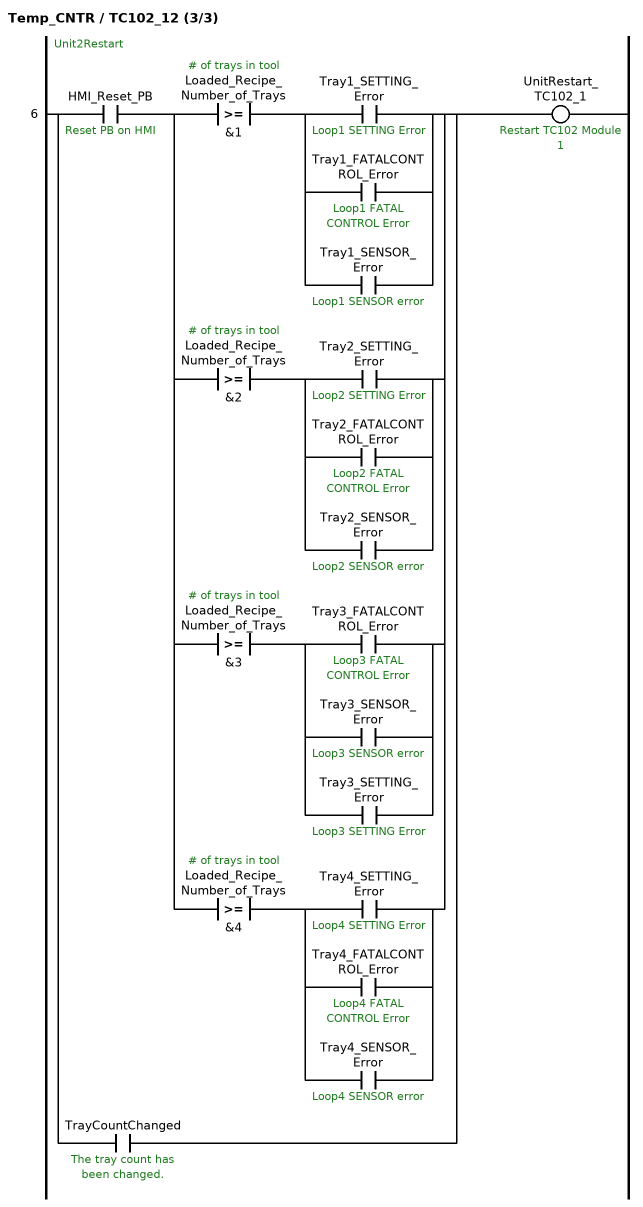
; rung 6: Unit2Restart
LD HMI_Reset_PB  ; Reset PB on HMI
LD>=(325) Loaded_Recipe_Number_of_Trays &1  ; # of trays in tool
LD Tray1_SETTING_Error  ; Loop1 SETTING Error
OR Tray1_FATALCONTROL_Error  ; Loop1 FATAL CONTROL Error
OR Tray1_SENSOR_Error  ; Loop1 SENSOR error
ANDLD
LD>=(325) Loaded_Recipe_Number_of_Trays &2  ; # of trays in tool
LD Tray2_SETTING_Error  ; Loop2 SETTING Error
OR Tray2_FATALCONTROL_Error  ; Loop2 FATAL CONTROL Error
OR Tray2_SENSOR_Error  ; Loop2 SENSOR error
ANDLD
ORLD
LD>=(325) Loaded_Recipe_Number_of_Trays &3  ; # of trays in tool
LD Tray3_FATALCONTROL_Error  ; Loop3 FATAL CONTROL Error
OR Tray3_SENSOR_Error  ; Loop3 SENSOR error
OR Tray3_SETTING_Error  ; Loop3 SETTING Error
ANDLD
ORLD
LD>=(325) Loaded_Recipe_Number_of_Trays &4  ; # of trays in tool
LD Tray4_SETTING_Error  ; Loop4 SETTING Error
OR Tray4_FATALCONTROL_Error  ; Loop4 FATAL CONTROL Error
OR Tray4_SENSOR_Error  ; Loop4 SENSOR error
ANDLD
ORLD
ANDLD
OR TrayCountChanged  ; The tray count has been changed.
OUT UnitRestart_TC102_1  ; Restart TC102 Module 1

### Section TC102_34
; Unit 12, Input type 0, Dipswitch 1-2-3-4-5-6-7 Off,  8 On

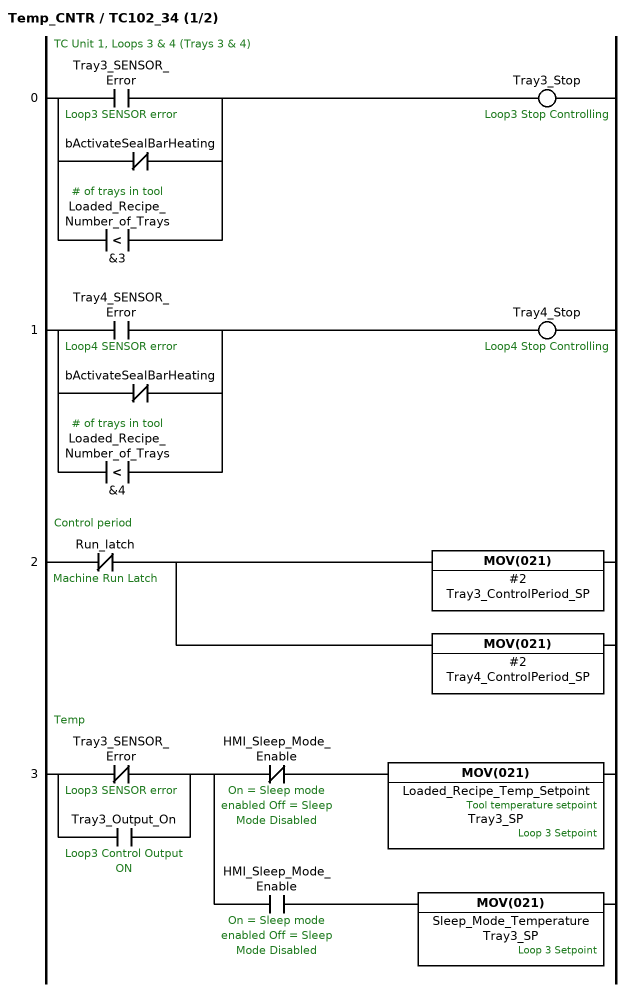
; rung 0: TC Unit 1, Loops 3 & 4 (Trays 3 & 4)
LD Tray3_SENSOR_Error  ; Loop3 SENSOR error
ORNOT bActivateSealBarHeating
OR<(310) Loaded_Recipe_Number_of_Trays &3  ; # of trays in tool
OUT Tray3_Stop  ; Loop3 Stop Controlling
; rung 1
LD Tray4_SENSOR_Error  ; Loop4 SENSOR error
ORNOT bActivateSealBarHeating
OR<(310) Loaded_Recipe_Number_of_Trays &4  ; # of trays in tool
OUT Tray4_Stop  ; Loop4 Stop Controlling
; rung 2: Control period
LDNOT Run_latch  ; Machine Run Latch
MOV(021) #2 Tray3_ControlPeriod_SP
MOV(021) #2 Tray4_ControlPeriod_SP
; rung 3: Temp
LDNOT Tray3_SENSOR_Error  ; Loop3 SENSOR error
OR Tray3_Output_On  ; Loop3 Control Output ON
OUT TR0
ANDNOT HMI_Sleep_Mode_Enable  ; On = Sleep mode enabled Off = Sleep Mode Disabled
MOV(021) Loaded_Recipe_Temp_Setpoint Tray3_SP  ; Tool temperature setpoint, Loop 3 Setpoint
LD TR0
AND HMI_Sleep_Mode_Enable  ; On = Sleep mode enabled Off = Sleep Mode Disabled
MOV(021) Sleep_Mode_Temperature Tray3_SP  ; Loop 3 Setpoint

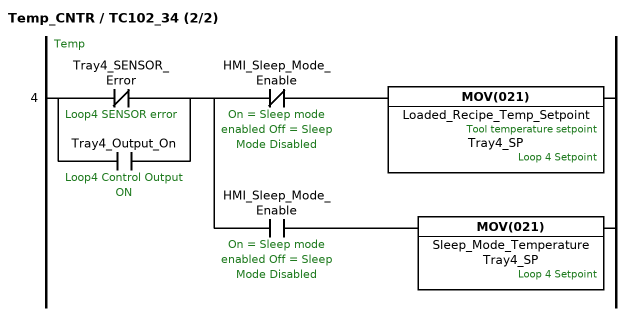
; rung 4: Temp
LDNOT Tray4_SENSOR_Error  ; Loop4 SENSOR error
OR Tray4_Output_On  ; Loop4 Control Output ON
OUT TR0
ANDNOT HMI_Sleep_Mode_Enable  ; On = Sleep mode enabled Off = Sleep Mode Disabled
MOV(021) Loaded_Recipe_Temp_Setpoint Tray4_SP  ; Tool temperature setpoint, Loop 4 Setpoint
LD TR0
AND HMI_Sleep_Mode_Enable  ; On = Sleep mode enabled Off = Sleep Mode Disabled
MOV(021) Sleep_Mode_Temperature Tray4_SP  ; Loop 4 Setpoint

### Section TC104_56

